TYPE TcoUrRobotics_T2O_State_IO : STRUCT
    bArray AT %I* : ARRAY[0..31] OF BYTE;
END_STRUCT
END_TYPE

(* stored: Version 1.1.0.1, ProductVersion 3.1.4024.12
   DUT TcoUrRobotics_T2O_State_IO: Id {162873de-b425-073d-00d6-f3dbdc611b62} *)
